Staubli VAL3: onF7Event.pgx

program onF7Event()
  local bool l_bYes
  local num l_nResult
  local string l_sMessage
begin
  if bButton[6] and sEvent!=""
    call deleteItem(l_bYes)
    if l_bYes
      call set:delete(sEvent,l_nResult)
      if l_nResult==0
        logMsg("[KERNEL] INTERFACE:Delete the box: "+" "+sEvent)
        call language2:message(l_sMessage,4)
        call use:timerDialog(l_sMessage,0)
        call set:onSave()
        call buildList()
      else
        popUpMsg("error code: "+toString("",l_nResult))
      endIf
    endIf
    call use:nullKey(nKey)
  endIf
end
